{attribute 'qualified_only'}
{attribute 'strict'}
{attribute 'to_string'}
TYPE E_DS402MoveMode :
(
    ABSOLUTE:=0,
    RELATIVE:=1
) UINT;
END_TYPE

(* stored: Version 1.1.0.1
   DUT E_DS402MoveMode: Id {e54849bb-1a7f-4171-a171-1e838b3e495e} *)
